TYPE CoeSettingData :
    STRUCT
    index             : UINT;
    subIndex          : BYTE;
    settingData       : POINTER TO INT;
    settingDataLength : UINT;
    settingLength     : UINT;
    END_STRUCT
END_TYPE

(* stored: Version 1.1.0.1, ProductVersion 3.1.4022.6
   DUT CoeSettingData: Id {a6982e9d-435b-4ac7-8f97-4ccbe30aa532} *)
